(* PLC project Unnamed, Unknown Unnamed 1 *)
(* stored: creationDateTime 2025-06-11T17:52:01, modificationDateTime 2025-06-12T18:54:32 *)

PROGRAM part3
  VAR
    CarSensor AT %IX0.0 : BOOL;
    PedButton AT %IX0.1 : BOOL;
    CarRedLight AT %QX0.0 : BOOL;
    CarYellowLight AT %QX0.1 : BOOL;
    CarGreenLight AT %QX0.2 : BOOL;
    PedRedLight AT %QX0.3 : BOOL;
    PedGreenLight AT %QX0.4 : BOOL;
  END_VAR
  VAR
    State : UINT := 0;
    wait_to_cross : UINT := 0;
    slow_cars : UINT := 1;
    ped_xing : UINT := 2;
    all_red : UINT := 3;
    SR0 : SR;
    TON0 : TON;
    TON1 : TON;
    TON2 : TON;
    reset_button : BOOL;
  END_VAR
  VAR  (* added by the conversion: wires and edge detectors of the diagram *)
    _EQ39_OUT : BOOL;
    _EQ4_OUT : BOOL;
    _EQ12_OUT : BOOL;
    _EQ25_OUT : BOOL;
    _MOVE36_ENO : BOOL;
    _MOVE36_OUT : UINT;
  END_VAR

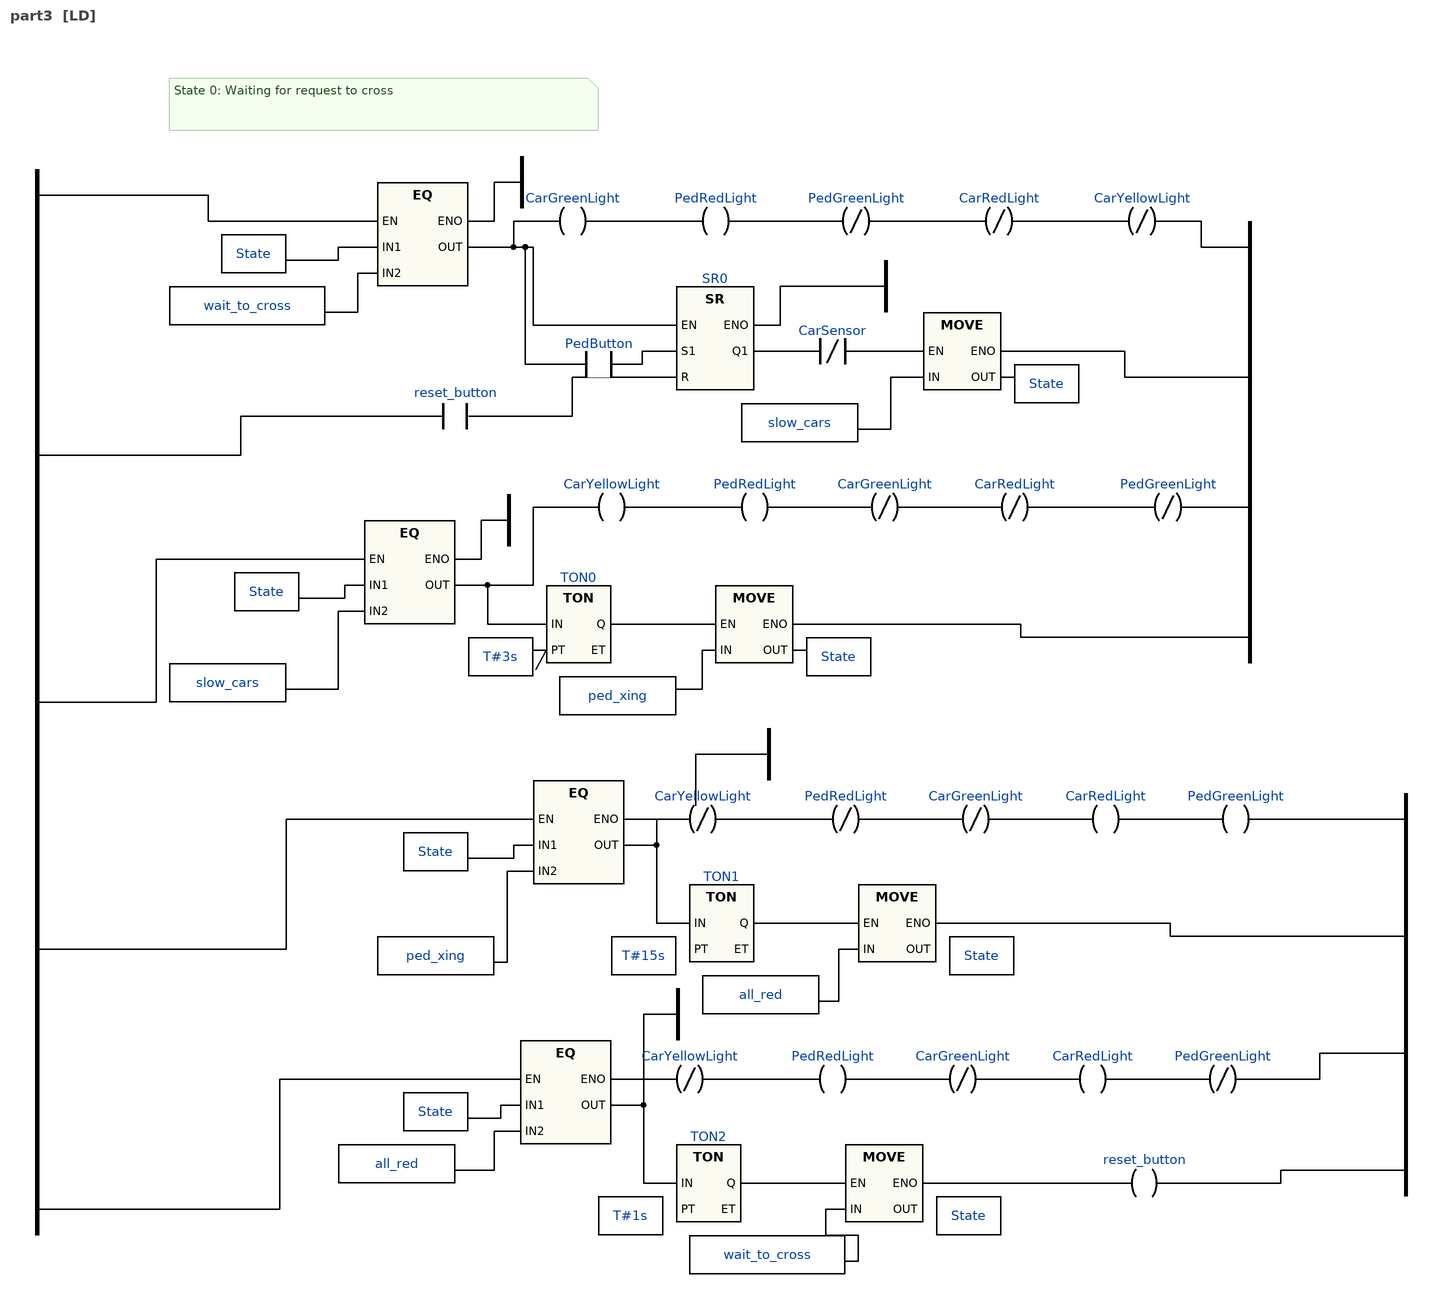
(* LD diagram, written out as Structured Text *)
(* State 0: Waiting for request to cross *)
_EQ39_OUT := State = wait_to_cross;
CarGreenLight := _EQ39_OUT;
PedRedLight := _EQ39_OUT;
SR0(EN := _EQ39_OUT, S1 := _EQ39_OUT AND PedButton, R := reset_button);
IF SR0.Q1 AND NOT CarSensor THEN State := slow_cars; END_IF;
_EQ4_OUT := State = slow_cars;
PedRedLight := _EQ4_OUT;
CarYellowLight := _EQ4_OUT;
TON0(IN := _EQ4_OUT, PT := T#3s);
IF TON0.Q THEN State := ped_xing; END_IF;
PedGreenLight := NOT _EQ39_OUT;
CarRedLight := NOT _EQ39_OUT;
CarYellowLight := NOT _EQ39_OUT;
CarGreenLight := NOT _EQ4_OUT;
CarRedLight := NOT _EQ4_OUT;
PedGreenLight := NOT _EQ4_OUT;
_EQ12_OUT := State = ped_xing;
CarYellowLight := NOT _EQ12_OUT;
PedRedLight := NOT _EQ12_OUT;
CarGreenLight := NOT _EQ12_OUT;
CarRedLight := _EQ12_OUT;
PedGreenLight := _EQ12_OUT;
_EQ25_OUT := State = all_red;
CarYellowLight := NOT _EQ25_OUT;
PedRedLight := _EQ25_OUT;
CarGreenLight := NOT _EQ25_OUT;
CarRedLight := _EQ25_OUT;
PedGreenLight := NOT _EQ25_OUT;
TON2(IN := _EQ25_OUT);
_MOVE36_OUT := MOVE(EN := TON2.Q, IN := wait_to_cross, ENO => _MOVE36_ENO);
reset_button := _MOVE36_ENO;
TON1(IN := _EQ12_OUT);
IF TON1.Q THEN MOVE(IN := all_red); END_IF;
(* drawn but not wired to any output: T#15s, T#1s *)
END_PROGRAM

CONFIGURATION Config0
  RESOURCE Res0 ON PLC
    TASK task0(INTERVAL := T#20ms, PRIORITY := 0);
    PROGRAM instance0 WITH task0 : part3;
  END_RESOURCE
END_CONFIGURATION
